{attribute 'qualified_only'}
VAR_GLOBAL
    stClamping : ST_ClampingProcessConfig := (bUseTorqueClamp := FALSE, bEnableMinClampTorqueCheck := FALSE, fMinClampTorquePercent := 0.0, fMaxClampTorquePercent := 30.0, tOverTorqueConfirm := T#200MS, stTorque := (fTargetTorquePercent := -20.0, fMaxAbsTorquePercent := 25.0, fTorqueRampPercentPerSecond := 50.0, fVelocityLimitHigh := 2.0, fVelocityLimitLow := -2.0, fReachedMinAbsTorquePercent := 16.0, tReachedStableTime := T#300MS, tTorqueBuildTimeout := T#3S, tModeSwitchTimeout := T#2S));
END_VAR
VAR_GLOBAL CONSTANT
    stTray : ST_TrayProcessConfig := (tLevelDetectStable := T#300MS);
    stVision : ST_VisionProcessConfig := (eMode := E_VisionMode.Camera, tDetectionDelay := T#2S, fSimulatedDetectedAngle := 60.0, fSimulatedCorrectionAngle := 60.0, bSimulatedDetected := TRUE, fSimulatedConfidence := 1.0, fAngleTolerance := 0.5);
    stCoaxVision : ST_CoaxVisionProcessConfig := (eVisionMode := E_VisionMode.Camera, fSimulatedCoaxiality := 0.0, fSimulatedDeltaX := 0.0, fSimulatedDeltaY := 0.0);
    stQrScan : ST_QrScanProcessConfig := (fOffsetAngle := 360.0);
    stGripper : ST_GripperProcessConfig := (tAcceptTimeout := T#3S, tResultTimeout := T#8S);
    stAdjustment : ST_AdjustmentProcessConfig := (fAdjustTolerance := 0.10, fQualifiedTolerance := 0.10,fMaxCorrectionX := 5.0,fMaxCorrectionY := 5.0, nMaxAdjustCount := 3, nMaxReworkCount := 1, nCoaxMaxRetryCount := 1, tCoaxRetryDelay := T#200MS);
    stScrewdriver : ST_ScrewdriverProcessConfig := (tPreTightenDuration := T#3S, tPreLoosenDuration := T#500MS, tFinalTightenDuration := T#3S, tReworkLoosenDuration := T#500MS);
END_VAR

(* stored: Version 1.1.0.1, ProductVersion 3.1.4026.20
   GVL GVL_ProcessConfig: Id {cf221c27-a9ba-43cd-a2d9-d3fb147708b7} *)
